(* IEC 61131-3 sources: Word/plc-course/11-program-organization/labs/starter, 3 files *)

(* ---- 11-1-motor-fb.st ---- *)
(* Lab 11-1: A reusable motor function block, used three times.
   Module 11 (Program organisation). STARTER - the FB interface, the program
   I/O and the three instances are declared for you. Write:
     1. the body of FB_Motor (and any internal variables it needs), and
     2. the program logic that calls Pump1, Pump2 and Fan1 and drives the outputs.
   Then run:
     python3 tools/plctest.py 11-program-organization/labs/starter/11-1-motor-fb.st *)

FUNCTION_BLOCK FB_Motor
  (* Direct-on-line motor with run feedback supervision.
     Keep these pin names: the test reads RunCmd, Running and Fault. *)
  VAR_INPUT
    Start       : BOOL;          (* start request, TRUE = start (pulse or held) *)
    Stop        : BOOL;          (* stop request, TRUE = stop; wins over Start *)
    InterlockOK : BOOL;          (* TRUE = allowed to run; FALSE stops the motor *)
    RunFb       : BOOL;          (* run feedback: contactor aux contact or airflow switch *)
    Reset       : BOOL;          (* fault reset *)
    FbTimeout   : TIME := T#2s;  (* how long RunFb may disagree with RunCmd *)
  END_VAR
  VAR_OUTPUT
    RunCmd      : BOOL;          (* command to the contactor coil *)
    Running     : BOOL;          (* proven running: RunCmd AND RunFb *)
    Fault       : BOOL;          (* latched feedback fault; needs Reset *)
    RunSeconds  : DINT;          (* optional extension (not tested): seconds of proven running *)
  END_VAR
  (* TODO: add a VAR ... END_VAR block here for internal variables,
     for example a TON instance for the feedback check. *)

  (* TODO: replace these placeholder lines with the motor logic. *)
  RunCmd := FALSE;
  Running := FALSE;
  Fault := FALSE;
END_FUNCTION_BLOCK

PROGRAM DosingRoom
  VAR (* inputs *)
    Pump1StartPB   AT %IX0.0 : BOOL;  (* Pump 1 start push-button, NO *)
    Pump1StopPB_NC AT %IX0.1 : BOOL;  (* Pump 1 stop push-button, NC: TRUE while not pressed *)
    Pump1RunFb     AT %IX0.2 : BOOL;  (* Pump 1 contactor auxiliary contact: TRUE = contactor in *)
    Pump2StartPB   AT %IX0.3 : BOOL;  (* Pump 2 start push-button, NO *)
    Pump2StopPB_NC AT %IX0.4 : BOOL;  (* Pump 2 stop push-button, NC *)
    Pump2RunFb     AT %IX0.5 : BOOL;  (* Pump 2 contactor auxiliary contact *)
    Fan1StartPB    AT %IX0.6 : BOOL;  (* Extract fan start push-button, NO *)
    Fan1StopPB_NC  AT %IX0.7 : BOOL;  (* Extract fan stop push-button, NC *)
    Fan1AirflowSw  AT %IX1.0 : BOOL;  (* Extract duct airflow switch: TRUE = air moving *)
    TankLowLow_NC  AT %IX1.1 : BOOL;  (* Day-tank low-low level switch, fail-safe:
                                         TRUE = level healthy, FALSE = low-low or wire break *)
    ResetPB        AT %IX1.2 : BOOL;  (* Fault reset push-button, NO *)
  END_VAR
  VAR (* outputs *)
    Pump1Contactor AT %QX0.0 : BOOL;  (* Pump 1 contactor coil *)
    Pump2Contactor AT %QX0.1 : BOOL;  (* Pump 2 contactor coil *)
    Fan1Contactor  AT %QX0.2 : BOOL;  (* Extract fan contactor coil *)
    FaultLamp      AT %QX0.3 : BOOL;  (* Common "motor fault" lamp *)
  END_VAR
  VAR (* one instance of FB_Motor per motor - keep these names *)
    Pump1 : FB_Motor;
    Pump2 : FB_Motor;
    Fan1  : FB_Motor;
  END_VAR

  (* TODO: call Fan1, Pump1 and Pump2 with the right inputs and parameters,
     then drive the contactors and the fault lamp from their outputs. *)
  Pump1Contactor := FALSE;
  Pump2Contactor := FALSE;
  Fan1Contactor := FALSE;
  FaultLamp := FALSE;
END_PROGRAM

CONFIGURATION Config0
  RESOURCE Res0 ON PLC
    TASK MainTask(INTERVAL := T#10ms, PRIORITY := 0);
    PROGRAM Inst0 WITH MainTask : DosingRoom;
  END_RESOURCE
END_CONFIGURATION

(* ---- 11-2-valve-fb.st ---- *)
(* Lab 11-2: A reusable on/off valve function block with limit switches.
   Module 11 (Program organisation). STARTER - the FB interface, the program
   I/O and the two instances are declared for you. Write:
     1. the body of FB_Valve (and any internal variables it needs), and
     2. the program logic that calls XV101 and XV102 and drives the outputs.
   Then run:
     python3 tools/plctest.py 11-program-organization/labs/starter/11-2-valve-fb.st

   XV101  reactor feed valve      fail CLOSED, 5 s travel time
   XV102  jacket cooling valve    fail OPEN,   8 s travel time
   Training exercise only: a real reactor trip belongs in a safety
   instrumented system, not in basic control logic (Module 20). *)

FUNCTION_BLOCK FB_Valve
  (* Single-solenoid, spring-return on/off valve with open and closed limit
     switches. Keep these pin names: the test reads IsOpen, IsClosed,
     TravelFault, LimitFault and Fault. *)
  VAR_INPUT
    OpenCmd    : BOOL;            (* TRUE = open, FALSE = close *)
    OpenLS     : BOOL;            (* open limit switch (ZSO), TRUE = fully open *)
    ClosedLS   : BOOL;            (* closed limit switch (ZSC), TRUE = fully closed *)
    Reset      : BOOL;            (* fault reset *)
    FailOpen   : BOOL;            (* configuration: TRUE = spring opens the valve *)
    TravelTime : TIME := T#10s;   (* longest acceptable stroke *)
  END_VAR
  VAR_OUTPUT
    Solenoid    : BOOL;           (* solenoid output *)
    IsOpen      : BOOL;           (* confirmed open *)
    IsClosed    : BOOL;           (* confirmed closed *)
    TravelFault : BOOL;           (* latched: did not reach / stay in position *)
    LimitFault  : BOOL;           (* latched: both limit switches made for 500 ms *)
    Fault       : BOOL;           (* TravelFault OR LimitFault *)
  END_VAR
  (* TODO: add a VAR ... END_VAR block here for internal variables
     (timers, the previous command, ...). *)

  (* TODO: replace these placeholder lines with the valve logic. *)
  Solenoid := FALSE;
  IsOpen := FALSE;
  IsClosed := FALSE;
  TravelFault := FALSE;
  LimitFault := FALSE;
  Fault := FALSE;
END_FUNCTION_BLOCK

PROGRAM ReactorValves
  VAR (* inputs *)
    XV101_OpenSw AT %IX0.0 : BOOL;  (* XV-101 panel selector: TRUE = OPEN, FALSE = CLOSE *)
    XV101_ZSO    AT %IX0.1 : BOOL;  (* XV-101 open limit switch *)
    XV101_ZSC    AT %IX0.2 : BOOL;  (* XV-101 closed limit switch *)
    XV102_OpenSw AT %IX0.3 : BOOL;  (* XV-102 panel selector: TRUE = OPEN, FALSE = CLOSE *)
    XV102_ZSO    AT %IX0.4 : BOOL;  (* XV-102 open limit switch *)
    XV102_ZSC    AT %IX0.5 : BOOL;  (* XV-102 closed limit switch *)
    ResetPB      AT %IX0.6 : BOOL;  (* Fault reset push-button, NO *)
  END_VAR
  VAR (* outputs *)
    XV101_SOL    AT %QX0.0 : BOOL;  (* XV-101 solenoid: energise to OPEN (fail closed) *)
    XV102_SOL    AT %QX0.1 : BOOL;  (* XV-102 solenoid: energise to CLOSE (fail open) *)
    FaultLamp    AT %QX0.2 : BOOL;  (* Common "valve fault" lamp *)
  END_VAR
  VAR (* device instances - keep these names *)
    XV101 : FB_Valve;               (* reactor feed valve *)
    XV102 : FB_Valve;               (* jacket cooling-water valve *)
  END_VAR

  (* TODO: call XV101 and XV102 with their inputs and configuration,
     then drive the solenoids and the fault lamp from their outputs. *)
  XV101_SOL := FALSE;
  XV102_SOL := FALSE;
  FaultLamp := FALSE;
END_PROGRAM

CONFIGURATION Config0
  RESOURCE Res0 ON PLC
    TASK MainTask(INTERVAL := T#10ms, PRIORITY := 0);
    PROGRAM Inst0 WITH MainTask : ReactorValves;
  END_RESOURCE
END_CONFIGURATION

(* ---- 11-3-function-library.st ---- *)
(* Lab 11-3: A small function library and a statistics FB using VAR_IN_OUT.
   Module 11 (Program organisation). STARTER - the record type, the function
   and FB interfaces and the program declarations are done for you. Write:
     1. the bodies of F_InRange and F_Deadband,
     2. the body of FB_SampleStats (and any internal variables it needs), and
     3. the program logic: clear, call Head1 and Head2, drive the reject
        gates and update ReportedMean.
   Then run:
     python3 tools/plctest.py 11-program-organization/labs/starter/11-3-function-library.st *)

TYPE
  ST_Stats :
  STRUCT
    Count    : DINT;    (* samples since the last clear *)
    InSpec   : DINT;    (* samples inside the limits *)
    OutSpec  : DINT;    (* samples outside the limits *)
    MinValue : REAL;    (* smallest sample since the last clear *)
    MaxValue : REAL;    (* largest sample since the last clear *)
    Sum      : LREAL;   (* running total (LREAL keeps precision over a long shift) *)
    Mean     : REAL;    (* Sum / Count *)
  END_STRUCT;
END_TYPE

FUNCTION F_InRange : BOOL
  (* TRUE when Low <= Value <= High (both limits included).
     If Low > High the range is empty: always FALSE. *)
  VAR_INPUT
    Value : REAL;
    Low   : REAL;
    High  : REAL;
  END_VAR
  (* TODO *)
  F_InRange := FALSE;
END_FUNCTION

FUNCTION F_Deadband : REAL
  (* Report-by-exception: return NewValue when it differs from OldValue by
     Band or more, otherwise return OldValue. *)
  VAR_INPUT
    NewValue : REAL;   (* live value *)
    OldValue : REAL;   (* value reported last time *)
    Band     : REAL;   (* smallest change worth reporting *)
  END_VAR
  (* TODO *)
  F_Deadband := 0.0;
END_FUNCTION

FUNCTION_BLOCK FB_SampleStats
  (* Adds one sample to the shared record Stats on each rising edge of
     Sample, and judges it against the limits with F_InRange.
     Keep these pin names: the test reads Reject and Samples. *)
  VAR_INPUT
    Sample    : BOOL;   (* rising edge = Value holds a new sample *)
    Value     : REAL;
    LowLimit  : REAL;
    HighLimit : REAL;
  END_VAR
  VAR_IN_OUT
    Stats     : ST_Stats;
  END_VAR
  VAR_OUTPUT
    Reject    : BOOL;   (* TRUE when this instance's latest sample was out of limits *)
    Samples   : DINT;   (* samples taken by THIS instance since power-up *)
  END_VAR
  (* TODO: add a VAR ... END_VAR block here for internal variables. *)

  (* TODO: replace this placeholder with the statistics logic. *)
  Reject := FALSE;
END_FUNCTION_BLOCK

PROGRAM CheckWeigher
  VAR (* inputs *)
    Head1Ready  AT %IX0.0 : BOOL;  (* check-weigher 1: TRUE when Head1Weight holds a new weight *)
    Head2Ready  AT %IX0.1 : BOOL;  (* check-weigher 2: TRUE when Head2Weight holds a new weight *)
    ClearPB     AT %IX0.2 : BOOL;  (* clear the line statistics (start of shift) *)
  END_VAR
  VAR (* outputs *)
    Head1Reject AT %QX0.0 : BOOL;  (* reject gate after head 1 *)
    Head2Reject AT %QX0.1 : BOOL;  (* reject gate after head 2 *)
  END_VAR
  VAR (* weights from the check-weighers and settings from the HMI *)
    Head1Weight  : REAL;             (* g, written by check-weigher 1 over the network *)
    Head2Weight  : REAL;             (* g, written by check-weigher 2 *)
    LowLimit     : REAL := 495.0;    (* g, lowest acceptable net weight *)
    HighLimit    : REAL := 505.0;    (* g, highest acceptable net weight *)
    MeanDeadband : REAL := 0.5;      (* g, smallest change of mean worth sending to SCADA *)
  END_VAR
  VAR (* data - keep these names *)
    LineStats    : ST_Stats;         (* shared by both heads, read by the HMI *)
    ReportedMean : REAL;             (* mean weight as last sent to SCADA *)
    Head1        : FB_SampleStats;
    Head2        : FB_SampleStats;
  END_VAR

  (* TODO: call Head1 and Head2 so that both update LineStats, keep every
     field of LineStats at zero while ClearPB is pressed (tip: a whole
     structure can be assigned in one statement; think about where in the
     scan to do it), drive the reject gates, and update ReportedMean with
     F_Deadband. *)
  Head1Reject := FALSE;
  Head2Reject := FALSE;
END_PROGRAM

CONFIGURATION Config0
  RESOURCE Res0 ON PLC
    TASK MainTask(INTERVAL := T#10ms, PRIORITY := 0);
    PROGRAM Inst0 WITH MainTask : CheckWeigher;
  END_RESOURCE
END_CONFIGURATION
